(* This testsuite creates a failed test with an empty assertion message *)
FUNCTION_BLOCK FB_EmptyAssertionMessage EXTENDS TcUnit.FB_TestSuite

IntegerEmptyAssertionMessage();

METHOD PRIVATE IntegerEmptyAssertionMessage
VAR
    a : INT := -32000;
    b : INT := 15423;
END_VAR
TEST('IntegerEmptyAssertionMessage');

AssertEquals_INT(Expected := a,
                 Actual := b,
                 Message := '');

TEST_FINISHED();
END_METHOD

END_FUNCTION_BLOCK

(* stored: Version 1.1.0.1, ProductVersion 3.1.4022.18
   POU FB_EmptyAssertionMessage: Id {d489f2ef-e9dc-4a48-95e4-bad84cbf1e42}, SpecialFunc None
   Method IntegerEmptyAssertionMessage: Id {993d3cc0-cd5a-4682-bc39-fee418867270} *)
